VAR_GLOBAL
		
//GVL_Devices
	{attribute 'pytmc' :=' pv: EM1K0:GEM:VCN:40 '}
	VCN_40 : FB_VCN;
	{attribute 'pytmc' :=' pv: EM1K0:GEM:VGP:40 '}
	VGP_40 : FB_VGP;
	
	{attribute 'pytmc' :=' pv: EM1K0:GEM:VVC:80 '}
	VVC_80:FB_VVC;
	{attribute 'pytmc' :=' pv: EM1K0:GEM:VVC:81 '}
	VVC_81:FB_VVC;
	{attribute 'pytmc' :=' pv: EM1K0:GEM:VVC:82 '}
	VVC_82:FB_VVC;
	{attribute 'pytmc' :=' pv: EM1K0:GEM:VVC:83 '}
	VVC_83 : FB_VVC;
	{attribute 'pytmc' :=' pv: EM1K0:GEM:VVC:84 '}
	VVC_84 : FB_VVC;
	{attribute 'pytmc' :=' pv: EM1K0:GEM:VVC:85 '}
	VVC_85 : FB_VVC;
	{attribute 'pytmc' :=' pv: EM1K0:GEM:VVC:86 '}
	VVC_86 : FB_VVC;
	

	{attribute 'pytmc' :=' pv: EM1K0:GEM:GCM:80 '}
	GCM_80: FB_GCM;
	
	{attribute 'pytmc' :=' pv: EM1K0:GEM:INJ_Override '}
	
	xOverrideMode : BOOL:= false;
		
//GVL_Sensors

(*Pressure Meter*)
	{attribute 'pytmc' :=' pv: EM1K0:GEM:GFM:86 '}
	GFM_86 :FB_PressureTransducer;
	{attribute 'pytmc' :=' pv: EM1K0:GEM:GFM:85 '}
	GFM_85 :FB_PressureTransducer;
	{attribute 'pytmc' :=' pv: EM1K0:GEM:GFM:84 '}
	GFM_84 :FB_PressureTransducer;
	{attribute 'pytmc' :=' pv: EM1K0:GEM:GFM:83 '}
	GFM_83 :FB_PressureTransducer;	

(*HV*)
	{attribute 'pytmc' :=' pv: EM1K0:GEM:HV:1 '}
	hv1 : FB_HighVoltage;
	{attribute 'pytmc' :=' pv: EM1K0:GEM:HV:2 '}
	hv2 : FB_HighVoltage;
	{attribute 'pytmc' :=' pv: EM1K0:GEM:RTD:1 '}
	RTD : FB_RTD;

END_VAR

(* stored: Version 1.1.0.1, ProductVersion 3.1.4022.12
   GVL GVL_INJ: Id {b0e309d1-2282-43cb-a77d-1c68f1ea549b} *)
